PROGRAM testFlexiBuffer
VAR
	shelf : Shelf(2, 2);
	shelfElements: ARRAY[0..100] OF ShelfElement;
	
	flexibuf: FlexiBuffer;
	state: TestFlexiBufferState;
	
	shelfElement: IShelfElement;
	
	usedElementsCount: UINT := 0;
	i: UINT;
END_VAR


shelf.getNextFreeSpace();

CASE state OF
TestFlexiBufferState.INIT:
	FOR i:=0 TO 3 DO
		usedElementsCount := usedElementsCount + 1;
		flexibuf.addElement(shelfElements[usedElementsCount - 1]);
	END_FOR;
	state := TestFlexiBufferState.WAIT;
	
TestFlexiBufferState.ADD_ELEMENT:
	usedElementsCount := usedElementsCount + 1;	
	flexibuf.addElement(shelfElements[usedElementsCount-1]);	
	state := TestFlexiBufferState.WAIT;

TestFlexiBufferState.REMOVE_ELEMENT:
	shelfElement := flexibuf.removeFirstElement();
	state := TestFlexiBufferState.WAIT;
	
END_CASE

END_PROGRAM

(* stored: Version 1.1.0.1
   POU testFlexiBuffer: Id {ac9acdb8-d283-4f96-994f-f9fabf800948}, SpecialFunc None *)
